PROGRAM TempPID
VAR
	
	PIDCooling: FB_BasicPID;
	PIDHeating: FB_BasicPID;
	bResetCooling: BOOL;
	bResetHeat: BOOL;

END_VAR

VAR_OUTPUT
	CoolingOutput: LREAL;
	HeatingOutput: LREAL;
END_VAR



//Run pid loop
PIDCooling(
	fSetpointValue:=GVL.TempSetpoint,
	fActualValue:=GVL.Temp, 
	bReset:=bResetCooling, 
	fCtrlCycleTime:=1, 
	fKp:=GVL.KpCooling, 
	fTn:=GVL.KiCooling, 
	fTv:=GVL.KvCooling, 
	fTd:=GVL.KdCooling);



PIDHeating(
	fSetpointValue:=GVL.TempSetpoint,
	fActualValue:=GVL.Temp, 
	bReset:=bResetHeat, 
	fCtrlCycleTime:=1, 
	fKp:=GVL.KpHeating - ((GVL.Light1Percent + GVL.Light2Percent)/GVL.lightLoad)*GVL.KpHeating, //If the lights are on, you really don't need that much heating. So we scale it back based on how many lights are on.
	fTn:=GVL.KiHeating, 
	fTv:=GVL.KvHeating, 
	fTd:=GVL.KdHeating);
	
//Reset the PID back to 0 if the output is out of range
IF  PIDCooling.fCtrlOutput>GVL.valveDeadZone OR PIDCooling.fCtrlOutput<-999999999 THEN
	bResetCooling:=TRUE;
	CoolingOutput:=0;
ELSIF GVL.reset =  TRUE THEN
	bResetCooling:=TRUE;
	
ELSE
	bResetCooling:=FALSE;	
	CoolingOutput:=PIDCooling.fCtrlOutput*-1+GVL.valveDeadZone;//<----important scaling function because the old staefa valves are weird. See documentation for siemens ZM-101A
END_IF

//Reset the PID back to 0 if the output is out of range
IF PIDHeating.fCtrlOutput<0 OR PIDHeating.fCtrlOutput>999999999 THEN
	bResetHeat:=TRUE;
ELSIF GVL.reset =  TRUE THEN
	bResetHeat:=TRUE;
ELSE
	bResetHeat:=FALSE;
	HeatingOutput:=PIDHeating.fCtrlOutput;
END_IF

//If there is a lot of cooling demand, turn off the heaters completely. (i.e. don't waste energy)
IF PIDCooling.fCtrlOutput<-2000 THEN
	HeatingOutput:=0;
END_IF




//Scale temp signal for analog out to avoid overflows/negative numbers
IF CoolingOutput>=32767 THEN
	GVL.iTempControl :=32767;
ELSIF CoolingOutput <=0 THEN
	GVL.iTempControl :=0;
ELSE
	GVL.iTempControl := LREAL_TO_INT(CoolingOutput);
END_IF

IF HeatingOutput>=30000 THEN
	HeatingOutput :=30000;
ELSIF HeatingOutput <=0 THEN
	HeatingOutput :=0;
ELSE
	HeatingOutput := HeatingOutput;
END_IF

END_PROGRAM

(* stored: Version 1.1.0.1, ProductVersion 3.1.4022.18
   POU TempPID: Id {3c95c5e7-09a7-440b-8471-771a74e09587}, SpecialFunc None *)
